PROGRAM MAIN
VAR
	fbPower: MC_POWER;
	biLimFwd AT %I*: BOOL;
	biLimBwd AT %I*: BOOL;
	boBrake AT %Q*:BOOL;
	bEnable: BOOL := TRUE;
	bHalt AT %Q*: BOOL ;
END_VAR


LadderLogic();

Axis1();
Axis2();
Axis3();
Axis4();
Axis5();
Axis6();

Axis7();
Axis8();
Axis9();
Axis10();

END_PROGRAM

(* stored: Version 1.1.0.1, ProductVersion 3.1.4022.3
   POU MAIN: Id {8732fc72-5f01-4166-8591-38c357bf3993}, SpecialFunc None *)
